INTERFACE ITF_Car

PROPERTY p_Locked : BOOL
GET
END_GET
SET
END_SET
END_PROPERTY

END_INTERFACE

(* stored: Version 1.1.0.1, ProductVersion 3.1.4024.12
   Itf ITF_Car: Id {db28b9c9-9ce4-4367-9c76-e0097f42a943}
   Property p_Locked: Id {73bd7050-5fa0-41ec-aacc-eb94aaf2fedf}
   Get Get: Id {cf8d8e33-dd2e-4565-a438-5937e84b0a47}
   Set Set: Id {ed1c8819-440a-4240-9147-3447aab7e354} *)
